FUNCTION_BLOCK FB_TopMold
VAR CONSTANT
	sCycleStateTextDef: ARRAY[0..25]  OF STRING :=	
		['State 0: Wait for Start',
		'State 1: Wait for signal to start move down',
		'State 2: Move down',
		'State 3: Drying lock time, Building pressure',
		'State 4: Start drying time',
		'State 5: Open pressure relief valve',
		'State 6: Vacuum time closed',
		'State 7: Move up',
		'State 8: Wait until take out unit is moving up and start blowoff',
		'State 9: Await blowoff time and stop blowoff',
		'State 10:',
		'State 11:',
		'State 12:',
		'State 13:',
		'State 14:',
		'State 15:',
		'State 16:',
		'State 17:',
		'State 18:',
		'State 19:',
		'State 20: Stop cycle state',																
		'State 21: Stop cycle state',
		'State 22:',
		'State 23:',
		'State 24:',
		'State 25:Stop direct state'];
	
	tCycleStateTimeouts: ARRAY[0..10] OF TIME := 
		[T#10S,T#10S,T#10S,T#10S,T#10S,T#10S,T#10S,T#10S,T#10S,T#10S,
		T#10S];

	sInitStateTextDef: ARRAY[0..10] OF STRING :=
		['State 0: Wait for Init Start',
		'State 1: Await pressure relief',
		'State 2: Move up',
		'State 3: Description Init State 3',
		'State 4: Description Init State 4',
		'State 5: Description Init State 5',
		'State 6: Description Init State 6',
		'State 7: Description Init State 7',
		'State 8: Description Init State 8',
		'State 9: Description Init State 9',
		'State 10: Stop init state'];

	tInitStateTimeouts: ARRAY[0..10] OF TIME := 
		[T#10S,T#10S,T#10S,T#10S,T#10S,T#10S,T#10S,T#10S,T#10S,T#10S
		,T#10S];
END_VAR

VAR_INPUT
	mxReset							: BOOL;	(*Reset Error*)
	mxEmergency						: BOOL;
	mxDoorsOpened					: BOOL;
	mxAutoMode						: BOOL; (* TRUE = Automode *)
	mxEmptyMachine					: BOOL;
	mxEnableHeating					: BOOL;

	mxResetCycleState				: BOOL;
	mxResetInitState				: BOOL;


	mxMoveUp						: BOOL; (* Drying finished or transfer ready with new product *)
	mxTakeOutIsMovingUp				: BOOL;
	ActualPositionTransfermold		: REAL;
	RHSR_Blocked 					: BOOL;
	
	(*Signals*)
	sgMoveDown						: BOOL; (* Signal from bottommold *)
END_VAR
VAR_IN_OUT
	MachParameters					: ST_TopMoldMachPar;
	ProdParameters					: ST_TopMoldProdPar;
END_VAR
VAR_OUTPUT
(*Errors*)
	Errors							: ST_TopMoldErrors;
	mxErrorInit						: BOOL;		(* Error, stop immediately. Initialisation neccesary *)
	mxErrorStopinPos				: BOOL;		(* Error, stop in position. Only reset neccesary *)

(* State vars *)
	mxCycleBusy						: BOOL;
	mxInitBusy						: BOOL;
	
(* Vars *)
	mxInitialized					: BOOL;
	

	mxCilIsMovingIn					: BOOL;
	mxCilIsMovingOut				: BOOL;
	mxCilIsIn						: BOOL;
	mxCilIsOut						: BOOL;	
	ActualPosition					: REAL;
	
(*Signals*)
	SgTmIsUp						: BOOL;	// Signals that the topmold is up
	SgTmIsDown						: BOOL; // Signals that the topmold is down
	
END_VAR
VAR
(* State vars *)
	miCycleState					: INT :=0;
	miCycleOldstate					: INT :=0;
	mxCycleTransitionState			: BOOL := FALSE;
	sCycleStateText					: STRING;
	exCycleTimeOut					: BOOL;		(* Timeout for the whole programcycle *)
	CycleTimeout					: TON;
	CycleTimeOutUpFlank				: R_TRIG;
	mxCycleTimeoutEnable			: BOOL;
	CycleTime						: REAL;
	mxCycleHasError					: BOOL;
	miStopState						: INT;
	mxStartCycle					: BOOL;
	mxStopCycle						: BOOL;
	mxStopDirect					: BOOL;
	
	miInitState						: INT	:=0;
	miInitOldstate					: INT	:=0;
	mxInitTransitionState			: BOOL	:= FALSE;
	sInitStateText					: STRING;
	exInitTimeOut					: BOOL;		(* Timeout for the whole programcycle *)
	InitTimeout						: TON;
	InitTimeOutUpFlank				: R_TRIG;
	mxInitTimeoutEnable				: BOOL;
	InitTime						: REAL;
	mxInitHasError					: BOOL;
	mxStartInit						: BOOL;
	mxStopInit						: BOOL;
(* Objects *)
	HydraulicCilinder				: FB_HydraulicCilinderAnalog;
	Vacuum							: FB_MonoValveNoFdbck;
	BlowOff							: FB_MonoValveNoFdbck;
	HeatingZone						: ARRAY [1..6] OF FB_Heatingzone;
(* Vars *)
	T_DryingTime					: TON;
	T_BlowOffClosed					: TON;
	RT_TakeOutIsMovingUp			: R_TRIG;
	T_DryingMoldLock				: TON;
	T_VacuumTimeClosed				: TON;
	T_BlowOff						: TON;
	RT_EnableBlowOff				: R_TRIG;
	RT_EnableVacuum					: R_TRIG;
	RT_StartBlowOffClosed: R_TRIG;
	RT_StartVacuumClosed: R_TRIG;
	T_StartVacuumAfterDrying: TON;
	RT_StartVacuumAfterDrying: R_TRIG;
	TestTime: TIME := T#24500MS;
END_VAR

Error();
Init();
Cycle();
Objects();

ActualPosition := HydraulicCilinder.ActPosition;

{region "Closed vacuum and blowoff HMI stuff"}
RT_EnableBlowOff(CLK:=MachParameters.EnableClosedBlowOff);
RT_EnableVacuum(CLK:=MachParameters.EnableClosedVacuum);

IF RT_EnableBlowOff.Q THEN
	MachParameters.EnableClosedVacuum := FALSE;
END_IF

IF RT_EnableVacuum.Q THEN
	MachParameters.EnableClosedBlowOff := FALSE;
END_IF
{endregion}

ACTION Cycle:
(*StateChange (Transition)  Signalgeneration*)
mxCycleTransitionState:=(miCycleState<>miCycleOldstate);
(*State text*)
sCycleStateText:=sCycleStateTextDef[miCycleState];
(*Timeout Watchdog for Statemachine*)
mxCycleTimeoutEnable:=NOT (miCycleState=0) AND NOT mxReset;

CycleTimeout(IN:=mxCycleTimeoutEnable  , PT:=tCycleStateTimeouts[miCycleState] );
CycleTimeOutUpFlank(CLK:=CycleTimeout.Q );
miCycleOldstate:=miCycleState;

(*Set Errorbit when Raising edge of Timeout has been detected*)
IF CycleTimeOutUpFlank.Q THEN
	exCycleTimeOut:=TRUE; 			(* 1 Timeout for the whole programcycle *)
END_IF

(*Function to reset the Statemachine*)
IF mxResetCycleState THEN
	mxResetCycleState:= FALSE;
	mxInitialized := FALSE;
		
	miCycleState:=0;
	miCycleOldstate:=miCycleState;
	mxCycleTransitionState:=FALSE;

	mxStartCycle:= FALSE;
	mxStopCycle:= FALSE;
	mxStopDirect:=FALSE;
	SgTmIsDown := FALSE;
	SgTmIsUp := FALSE;
	mxMoveUp := FALSE;
	sgMoveDown := FALSE;

	T_DryingTime.IN:= FALSE;
	T_DryingMoldLock.IN:= FALSE;
	T_VacuumTimeClosed.IN:= FALSE;
	T_BlowOffClosed.IN:= FALSE;
	T_BlowOff.IN:=FALSE;	
	
	HydraulicCilinder.M_Stop();
END_IF

// Test CODE!
//RT_StartVacuumAfterDrying(CLK:=(miCycleState = 4));
//T_StartVacuumAfterDrying(IN:=, PT:=TestTime);
(*
IF RT_StartVacuumAfterDrying.q THEN
	T_StartVacuumAfterDrying.IN:=TRUE;
END_IF

IF T_StartVacuumAfterDrying.q THEN
	T_StartVacuumAfterDrying.IN := FALSE;
	Vacuum.M_On();
END_IF
*)

(*Definition State has Error*)
mxCycleHasError:=FALSE;

T_BlowOff(IN:=, PT:=MachParameters.BlowOffToTakeOut);
T_DryingTime(IN:= , PT:= MachParameters.DryingTime);

{region "Vacuum / Blowoff while closed"}
	T_VacuumTimeClosed(IN:= , PT:= MachParameters.VacuumTimeClosed);
	T_BlowOffClosed(IN:= , PT:= MachParameters.BlowOffTimeClosed);
	RT_StartBlowOffClosed(CLK:= MachParameters.EnableClosedBlowOff AND (miCycleState = 4));
	RT_StartVacuumClosed(CLK:=MachParameters.EnableClosedVacuum AND (miCycleState = 4));
	
	IF RT_StartBlowOffClosed.Q THEN 
		T_BlowOffClosed.IN := TRUE;
		BlowOff.M_On();
	ELSIF RT_StartVacuumClosed.Q THEN
		T_VacuumTimeClosed.IN := TRUE;
		Vacuum.M_On();
	END_IF
	
	IF T_BlowOffClosed.Q THEN 
		T_BlowOffClosed.IN := FALSE;
		BlowOff.M_Off(); 
	END_IF
	IF T_VacuumTimeClosed.Q THEN 
		T_VacuumTimeClosed.IN := FALSE;
		Vacuum.M_Off(); 
	END_IF
{endregion}


(*Cycle State's*)
CASE miCycleState OF

{region "Description"}
	(* Cycle:
	LEEG beginnen
		-wacht op signaal vanuit bottommold, naar beneden
		-Naar beneden om product te drogen
		-als bijna dicht dan extra druk opbouwen
		-Na droogtijd/transfer up wait time, relief presure
		-vacuum aan, omhoog, signal to bottom mold -> vac of blow on
		-signaal Mold is up -> bottom mold
		-Wacht op bottom mold is in
		-Wacht op takeout unit is omhoog (als enabled)
		-blow off aan*)
{endregion}
	0:
		IF mxStartCycle THEN
			mxStartCycle:= FALSE;
			miCycleState:= 1;
		END_IF
	
	1: // wait for move down
		
		// Keep topmold in its "up" position.
		HydraulicCilinder.M_Move(EndPosition:= MachParameters.PositionUpStop,  NormalSpeed:= MachParameters.SpeedUpNormal, 
								SlowPosition:= MachParameters.PositionUpStop - MachParameters.PositionUpSlow, SlowSpeed:= MachParameters.SpeedUpSlow, 
								CreepPosition:=MachParameters.PositionUpStop - MachParameters.PositionUpCreep, CreepSpeed:=MachParameters.SpeedUpCreep);
 
		IF mxStopDirect THEN
			mxStopDirect:= FALSE;
			miCycleState:= 25;
		ELSIF mxStopCycle AND mxEmptyMachine THEN
			mxStopCycle:=False;
			mxEmptyMachine:= FALSE;
			miCycleState:= 0;
		ELSIF mxStopCycle THEN
			mxStopCycle:= FALSE;
			miStopState:= miCycleState;
			miCycleState:= 0;
		ELSIF sgMoveDown THEN	
			sgMoveDown:= FALSE;
			mxMoveUp:= FALSE;
			SgTmIsUp:= FALSE;
			miCycleState:= 2;
		END_IF
			
	2: // Move down. 
		IF mxStopDirect THEN
			mxStopDirect:= FALSE;
			miCycleState:= 25;(*Stop direct*)
		ELSIF mxStopCycle THEN
			mxStopCycle:= FALSE;
			miStopState:= miCycleState;
			miCycleState:= 20;
		ELSIF HydraulicCilinder.M_Move(EndPosition:=ProdParameters.PositionDownStop, NormalSpeed:=MachParameters.SpeedDownNormal, 
										SlowPosition:=ProdParameters.PositionDownStop + Machparameters.PositionDownSlow, SlowSpeed:=MachParameters.SpeedDownSlow, 
										CreepPosition:=ProdParameters.PositionDownStop + Machparameters.PositionDownCreep, CreepSpeed:=MachParameters.SpeedDownCreep) THEN
			//BlowOff.M_On(); 			// Blowoff stops after delay ^ at top of cylce
			miCycleState:= 3;
		END_IF
	
	3: // Drying Lock time, build up pressure 
		IF mxStopDirect THEN
			mxStopDirect:= FALSE;
			miCycleState:= 25;(*Stop direct*)
		ELSIF mxStopCycle THEN
			mxStopCycle:= FALSE;
			miStopState:= miCycleState;
			miCycleState:= 20;
		ELSIF TRUE  THEN 	// ELSIF HydraulicCilinder.M_Press(Pressdown:=TRUE, PressSpeed:=MachParameters.PressSpeed, StoppingPressure:=MachParameters.PressStop) THEN
			//HydraulicCilinder.M_Stop();		
			sgTmIsDown:= TRUE;
			sgTmIsUp:=FALSE;
			miCycleState:= 4;
		END_IF
	
	
	4:  // start drying 
		T_DryingTime(IN:= TRUE);
		
		HydraulicCilinder.M_Press(Pressdown:=TRUE, PressSpeed:=MachParameters.PressSpeed, StoppingPressure:=MachParameters.PressStop);
		
		IF mxStopDirect THEN
			mxStopDirect:= FALSE;
			miCycleState:= 25;(*Stop direct*)
		ELSIF mxStopCycle THEN
			mxStopCycle:= FALSE;
			miStopState:=miCycleState;
			miCycleState:= 20;
		ELSIF T_DryingTime.Q THEN		// When dryingtime has finished, allways open up
			T_DryingTime(IN:= FALSE);
			Vacuum.M_On();
			miCycleState:= 5;
		END_IF
		
	5: // Move up to "open" position with "slow" speed 
		IF mxStopDirect THEN
			mxStopDirect:= FALSE;
			miCycleState:= 25;
		ELSIF mxStopCycle THEN
			mxStopCycle:= FALSE;
			miStopState:= miCycleState;
			miCycleState:= 20;
		ELSIF HydraulicCilinder.M_Move(EndPosition:= ProdParameters.PositionDownOpen,  NormalSpeed:=MachParameters.SpeedOpening, 
										SlowPosition:= ProdParameters.PositionDownOpen, SlowSpeed:=MachParameters.SpeedOpening, 
										CreepPosition:=ProdParameters.PositionDownOpen, CreepSpeed:=MachParameters.SpeedOpening) THEN
			miCycleState:= 6;
		END_IF
	
		
	6: // Move up 
		IF mxStopDirect THEN
			mxStopDirect:= FALSE;
			miCycleState:= 25;
		ELSIF mxStopCycle THEN
			mxStopCycle:= FALSE;
			miStopState:= miCycleState;
			miCycleState:= 20;
		ELSIF HydraulicCilinder.M_Move(EndPosition:= MachParameters.PositionUpStop,  NormalSpeed:= MachParameters.SpeedUpNormal, 
										SlowPosition:= MachParameters.PositionUpStop - MachParameters.PositionUpSlow, SlowSpeed:= MachParameters.SpeedUpSlow, 
										CreepPosition:=MachParameters.PositionUpStop - MachParameters.PositionUpCreep, CreepSpeed:=MachParameters.SpeedUpCreep) THEN
			SgTmIsUp:= TRUE;
			SgTmIsDown:= FALSE;
			mxMoveUp:= FALSE;
			
			miCycleState:= 7;
		END_IF
		
	7: //Wait until takeout is moving up *)	
	
		IF mxStopDirect THEN
			mxStopDirect:= FALSE;
			miCycleState:= 25;(*Stop direct*)
		ELSIF mxStopCycle THEN
			mxStopCycle:= FALSE;
			HydraulicCilinder.M_Stop();
			miStopState:= miCycleState;
			miCycleState:= 20;
		ELSIF mxTakeOutIsMovingUp THEN
			Vacuum.M_Off();
			BlowOff.M_On();
			
			miCycleState:= 8;
		END_IF
		
	8: // Await Blowoff
		T_BlowOff.IN := TRUE;
		
		IF mxStopDirect THEN
			mxStopDirect:= FALSE;
			miCycleState:= 25;(*Stop direct*)
		ELSIF mxStopCycle THEN
			mxStopCycle:= FALSE;
			HydraulicCilinder.M_Stop();
			miStopState:= miCycleState;
			miCycleState:= 20;
		ELSIF T_BlowOff.Q THEN
			BlowOff.M_Off();
			
			T_BlowOff.IN := FALSE;
			miCycleState:= 1;
		END_IF

	20: // Stop Cycle
		IF mxStopDirect THEN
			mxStopDirect:= FALSE;
			miCycleState:= 25;
		ELSIF TRUE THEN
			miCycleState:= 21;
		END_IF

	21:	//Stop cycle, wait for start
		IF mxStopDirect THEN
			mxStopDirect:= FALSE;
			miCycleState:= 25;
		ELSIF mxStartCycle THEN

			miCycleState:= miStopState;
		END_IF
	(* Stop Direct *)	
	25:
		mxStartCycle:= FALSE;
		mxStopCycle:= FALSE;
		mxInitialized:= FALSE;

		T_DryingTime.IN:= FALSE;
		
		HydraulicCilinder.M_StopDirect();
		Vacuum.M_Off(); (* When product do not switch off *)
		BlowOff.M_Off();
	
		miCycleState:= 0;

END_CASE

mxCycleBusy:= miCycleState<>0 AND NOT (miCycleState=21);
END_ACTION

ACTION Error:


(* ****************************************************************************** *)
mxErrorStopInPos:= HydraulicCilinder.mxErrorStopInPos;
mxErrorInit:= HydraulicCilinder.mxErrorInit
			OR HeatingZone[1].mxErrorInit
			OR HeatingZone[2].mxErrorInit
			OR HeatingZone[3].mxErrorInit
			OR HeatingZone[4].mxErrorInit
			OR HeatingZone[5].mxErrorInit
			OR HEatingZone[6].mxErrorInit;
END_ACTION

ACTION Init:
(*StateChange (Transition)  Signalgeneration*)
mxInitTransitionState:=(miInitState<>miInitOldstate);
(*State text*)
sInitStateText:=sInitStateTextDef[miInitState];
(*Timeout Watchdog for Statemachine*)
mxInitTimeoutEnable:=NOT (miInitState=0)  AND NOT mxReset;

InitTimeout(IN:=mxInitTimeoutEnable  , PT:=tInitStateTimeouts[miInitState] );
InitTimeOutUpFlank(CLK:=InitTimeout.Q );
miInitOldstate:=miInitState;

(*Set Errorbit when Raising edge of Timeout has been detected*)
IF InitTimeOutUpFlank.Q THEN
	exInitTimeOut:=TRUE; 			(* 1 Timeout for the whole programcycle *)
END_IF

(*Function to reset the Statemachine*)
IF mxResetInitState THEN
	mxResetInitState:=FALSE;
	miInitState:=0;
	miInitOldstate:=miInitState;
	mxInitTransitionState:=FALSE;
	
	mxStartInit:= FALSE;
	mxStopInit:= FALSE;		
END_IF

(*Definition State has Error*)
mxInitHasError:=FALSE;

(*Init State's*)
CASE miInitState OF
	0:
		IF mxStartInit THEN
			mxStartInit:= FALSE;
			mxInitialized:=FALSE;
			
			Vacuum.M_Off();
			BlowOff.M_Off();

			miInitState:= 1;
		END_IF
		
	(* Move Up *)	
	1:
		IF mxStopInit THEN
			mxStopInit:= FALSE;

			miInitState:= 10;
		END_IF
			
		// Above Normal Position
		IF HydraulicCilinder.ActPosition > MachParameters.PositionUpStop THEN // Move down
			IF HydraulicCilinder.M_Move(EndPosition:=MachParameters.PositionUpStop, NormalSpeed:= MachParameters.SpeedUpNormal, 
											SlowPosition:=MachParameters.PositionUpStop + MachParameters.PositionUpSlow, SlowSpeed:=MachParameters.SpeedUpSlow, 
											CreepPosition:=MachParameters.PositionUpStop + MachParameters.PositionUpCreep,	CreepSpeed:=MachParameters.SpeedUpCreep ) THEN
			mxInitialized:= TRUE; (* Return val *)
			miInitState:= 0;	
			END_IF
		ELSE
		// Below normal position
			IF HydraulicCilinder.M_Move(EndPosition:=MachParameters.PositionUpStop, NormalSpeed:= MachParameters.SpeedUpNormal, 
											SlowPosition:=MachParameters.PositionUpStop - MachParameters.PositionUpSlow, SlowSpeed:=MachParameters.SpeedUpSlow, 
											CreepPosition:=MachParameters.PositionUpStop - MachParameters.PositionUpCreep,	CreepSpeed:=MachParameters.SpeedUpCreep ) THEN
			mxInitialized:= TRUE; (* Return val *)
			miInitState:= 0;	
			END_IF
		END_IF

	(* Stop Init *)
	10:
		HydraulicCilinder.M_Stop();

		mxStartInit:= FALSE;
		mxStopInit:= FALSE;
		mxInitialized:=FALSE;					

		miInitState:= 0;
END_CASE

mxInitBusy:= miInitState<>0;
END_ACTION

METHOD M_EmptyMachine

IF mxCycleBusy THEN
	mxEmptyMachine:= TRUE;	
END_IF
END_METHOD

METHOD M_StartCycle

IF NOT mxCycleBusy THEN
	mxStartCycle:= TRUE;	
	mxStopCycle := FALSE;
END_IF
END_METHOD

METHOD M_StartInit

IF NOT mxInitBusy THEN 
	mxStartInit:= TRUE; 
END_IF
END_METHOD

METHOD M_StopCycle

IF mxCycleBusy THEN 
	mxStopCycle:= TRUE; 
END_IF
END_METHOD

METHOD M_StopDirect

IF mxCycleBusy THEN
	mxStopDirect:= TRUE;	
END_IF
END_METHOD

METHOD M_StopInit

IF mxInitBusy THEN 
	mxStopInit:= TRUE; 
END_IF
END_METHOD

ACTION Objects:
(* Object Calls *)
HydraulicCilinder(
	mxReset:= mxReset, 
	mxEmergency:= mxEmergency OR mxDoorsOpened, 
	mxAutoMode:= mxAutoMode, 
	EndPositionIn:= MachParameters.PositionUpStop,
	EndPositionOut:= ProdParameters.PositionDownStop,
	OffsetPosition:= MachParameters.PositionOffsetZero,
	OffsetAlarmPosition:= MachParameters.PositionOffsetAlarm,
	PositionPhysicalMeasured:=MachParameters.PositionPhyscialMeasured,
	PositionPhysicalMeasuredOld:=MachParameters.PositionPhysicalMeasuredOld,
	PhysicalOffsetPos:=MachParameters.PhysicalOffsetPos,
	RHSR_Blocked:=RHSR_Blocked,
	mxIsMovingIn=> mxCilIsMovingIn, 
	mxIsMovingOut=> mxCilIsMovingOut, 
	ManSpeedCreepIn:=MachParameters.SpeedUpCreep,
	ManSpeedCreepOut:=MachParameters.SpeedDownCreep,
	ManSpeedSlowIn:=MachParameters.SpeedUpSlow,
	ManSpeedSlowOut:=MachParameters.SpeedDownSlow,
	ManSpeedIn:=MachParameters.SpeedUpNormal,
	ManSpeedOut:=MachParameters.SpeedDownNormal,
	mxIsIn=> mxCilIsIn, 
	mxIsOut=> mxCilIsOut,
	Errors=> Errors.Hydraulic);
	
Vacuum(
	mxReset:= mxReset, 
	mxEmergency:= mxEmergency OR mxDoorsOpened, 
	mxAutoMode:= mxAutoMode);
	
BlowOff(
	mxReset:= mxReset, 
	mxEmergency:= mxEmergency OR mxDoorsOpened, 
	mxAutoMode:= mxAutoMode);


HeatingZone[1](
	mxReset:= mxReset,
	mxEmergency:=mxEmergency,
	mxDoorsOpened:=mxDoorsOpened,
	mxEnableHeating:=mxEnableHeating,
	MachParameters:=MachParameters.HeatingZone[1],
	Errors=> Errors.HeatingZone[1]);
	
HeatingZone[2](
	mxReset:= mxReset,
	mxEmergency:=mxEmergency,
	mxDoorsOpened:=mxDoorsOpened,
	mxEnableHeating:=mxEnableHeating,
	MachParameters:=MachParameters.HeatingZone[2],
	Errors=> Errors.HeatingZone[2]);

HeatingZone[3](
	mxReset:= mxReset,
	mxEmergency:=mxEmergency,
	mxDoorsOpened:=mxDoorsOpened,
	mxEnableHeating:=mxEnableHeating,
	MachParameters:=MachParameters.HeatingZone[3],
	Errors=> Errors.HeatingZone[3]);

HeatingZone[4](
	mxReset:= mxReset,
	mxEmergency:=mxEmergency,
	mxDoorsOpened:=mxDoorsOpened,
	mxEnableHeating:=mxEnableHeating,
	MachParameters:=MachParameters.HeatingZone[4],
	Errors=> Errors.HeatingZone[4]);

HeatingZone[5](
	mxReset:= mxReset,
	mxEmergency:=mxEmergency,
	mxDoorsOpened:=mxDoorsOpened,
	mxEnableHeating:=mxEnableHeating,
	MachParameters:=MachParameters.HeatingZone[5],
	Errors=> Errors.HeatingZone[5]);

HeatingZone[6](
	mxReset:= mxReset,
	mxEmergency:=mxEmergency,
	mxDoorsOpened:=mxDoorsOpened,
	mxEnableHeating:=mxEnableHeating,
	MachParameters:=MachParameters.HeatingZone[6],
	Errors=> Errors.HeatingZone[6]);
END_ACTION

END_FUNCTION_BLOCK

(* stored: Version 1.1.0.1, ProductVersion 3.1.4022.16
   POU FB_TopMold: Id {2e250e61-b76c-4394-b65d-3dcc6d70421f}, SpecialFunc None
   Action Cycle: Id {aa84e275-3c1d-464c-ac84-bda18804604f}
   Action Error: Id {66da3a34-a24d-40b5-a841-1ea942d4ab90}
   Action Init: Id {f7aba8dc-4755-4b83-9e5d-3eeacad8d9cb}
   Method M_EmptyMachine: Id {427defab-33ee-46e3-b86c-26c43217307b}
   Method M_StartCycle: Id {60f5d12b-dd25-4393-b3b3-a2162a925419}
   Method M_StartInit: Id {1e7dd9cb-2b74-4360-92d5-d40cba4e6f74}
   Method M_StopCycle: Id {6b0e6f3c-2f7c-4e9c-b362-79a28a7b070e}
   Method M_StopDirect: Id {bb973ae9-b5f9-4eab-86c6-e4763c6aa73e}
   Method M_StopInit: Id {39a3f404-e2be-408d-b953-4425c44cc67f}
   Action Objects: Id {f4c6d122-9031-434d-b21e-1f3c62e81905} *)
